(* IEC 61131-3 sources: CodesysTest/alpha/export/Device.dev/Plc Logic/Application/ObjectHandling/FB_CollectionHandlerLogs.pou, 1 file *)

(* ---- FB_CollectionHandlerLogs.pou.st ---- *)
(*#-#-#-#-#-#-#-#-#-#---Declaration---#-#-#-#-#-#-#-#-#-#-#-#-#*)

FUNCTION_BLOCK FB_CollectionHandlerLogs
VAR_INPUT
END_VAR
VAR
	Collection: ARRAY[0..GlobalObjects.MAX_LOGS] OF IMachineLogger; // object array
	ObjNames   : ARRAY[0..GlobalObjects.MAX_LOGS] OF STRING;
	_ArrayOver   : BOOL;
	_BadObj      : INT;
	_DupeObj   : INT;
	_OverObj   : INT;
	_TotalObj   : UINT;
END_VAR(*#-#-#-#-#-#-#-#-#-#---Implementation---#-#-#-#-#-#-#-#-#-#-#-#-#*)
